FUNCTION_BLOCK FrameClass
VAR_INPUT
	AllFrames : ARRAY [0..20] OF StructFrame;
END_VAR
VAR_OUTPUT
END_VAR
VAR
END_VAR

METHOD DuplicateExists : INT
VAR_INPUT
	sTargetAlias : STRING;
END_VAR
VAR
	i : INT;
	n : INT;
END_VAR

FOR i := 0 TO 20 DO
	IF AllFrames[i].sAlias = sTargetAlias THEN
		n := i;
		EXIT;
	ELSE n:=0;
	END_IF
END_FOR

DuplicateExists := n;
END_METHOD

METHOD FindFirstEmpty : INT;
VAR_INPUT
END_VAR
VAR
	EmptyArr : ARRAY[0..20] OF StructFrame;
	i: INT;
	n: INT := 0;
END_VAR
FOR i:=1 TO 20 DO
	IF AllFrames[i].rXpos = 0.0 AND AllFrames[i].rYpos = 0.0 AND AllFrames[i].rZpos = 0.0 AND AllFrames[i].sAlias = '' THEN
		FindFirstEmpty := i;
		EXIT;
	END_IF
END_FOR
END_METHOD

METHOD GetNonEmptyFrameAlias : ARRAY [0..20] OF STRING;
VAR_INPUT
END_VAR
VAR
	i : INT;
	NonEmptyFrames : ARRAY [0..20] OF StructFrame;
	emptyArray : ARRAY [0..20] OF STRING;
END_VAR
NonEmptyFrames := NonEmpty();
FOR i := 0 TO 20 DO
	emptyArray[i] := NonEmptyFrames[i].sAlias;
END_FOR
GetNonEmptyFrameAlias := emptyArray;
END_METHOD

METHOD MapArrangedAliasToFrameIndex : ARRAY[0..20] OF StructFrame;
VAR_INPUT
	arrangedAlias : ARRAY [0..20] OF STRING;
	NonEmptyFrames : ARRAY [0..20] OF StructFrame;
END_VAR

VAR
	mappedArray : ARRAY [0..20] OF StructFrame;
	aliasIndex : INT;
	framesIndex : INT;
	arrangedIndex : INT := 0;
	emptyFrame : StructFrame;
END_VAR
FOR aliasIndex := 0 TO 20 DO
	IF arrangedAlias[aliasIndex] <>  'select' THEN
		FOR framesIndex := 0 TO 20 DO
			IF arrangedAlias[aliasIndex] = NonEmptyFrames[framesIndex].sAlias THEN
				mappedArray[arrangedIndex] := NonEmptyFrames[framesIndex];
				arrangedIndex := arrangedIndex + 1;
				EXIT;
			END_IF
		END_FOR
	ELSE
		mappedArray[arrangedIndex] := emptyFrame;
		arrangedIndex := arrangedIndex + 1;
	END_IF
END_FOR

MapArrangedAliasToFrameIndex := mappedArray;
END_METHOD

METHOD NonEmpty : ARRAY [0..20] OF StructFrame;
VAR_INPUT
END_VAR
VAR
	EmptyArray : ARRAY [0..20] OF StructFrame;
	i : INT;
	n : INT := 0;
END_VAR
FOR i:=1 TO 20 DO
	IF NOT (AllFrames[i].rXpos = 0.0) AND NOT (AllFrames[i].rYpos = 0.0) AND NOT (AllFrames[i].rZpos = 0.0) THEN
		EmptyArray[n] := AllFrames[i];
		n := n+1;
	END_IF
END_FOR
NonEmpty := EmptyArray;
END_METHOD

METHOD Teach : BOOL
VAR_INPUT
	iArrayIndex : INT;
	rCurrentXpos : REAL;
	rCurrentYpos : REAL;
	rCurrentZpos : REAL;
	sAlias : STRING;
END_VAR
VAR
	bSuccess : BOOL := FALSE;
	AugmentedFrame : StructFrame;
END_VAR
AllFrames[iArrayIndex].rXpos := rCurrentXpos;
AllFrames[iArrayIndex].rYpos := rCurrentYpos;
AllFrames[iArrayIndex].rZpos := rCurrentZpos;
AllFrames[iArrayIndex].sAlias := sAlias;
Teach := TRUE;
END_METHOD

END_FUNCTION_BLOCK

(* stored: Version 1.1.0.1, ProductVersion 3.1.4024.9
   POU FrameClass: Id {494de9e0-eb30-4118-9b19-660d2a4d7b01}, SpecialFunc None
   Method DuplicateExists: Id {4c0d7f0f-c44b-4de5-9f9f-1a7ee1126f00}
   Method FindFirstEmpty: Id {dbc83be6-9e01-48c0-bed1-c73635c56031}
   Method GetNonEmptyFrameAlias: Id {ecabe442-790f-435a-9e97-b1468f072709}
   Method MapArrangedAliasToFrameIndex: Id {85f5c58b-a959-4faf-ad1b-28794b23e3ad}
   Method NonEmpty: Id {7514c85b-d3cb-4aaf-a59d-4aec763a260f}
   Method Teach: Id {cb1dc23b-6b3f-4e2b-89ef-3a06cf855ec7} *)
